FUNCTION_BLOCK FB_LightOffCommand IMPLEMENTS I_Command
VAR_INPUT
END_VAR
VAR_OUTPUT
END_VAR
VAR
	// Reference to the Light that should be switched on.
	iLight: I_Switchable;
END_VAR

METHOD Execute
IF (iLight <> 0) THEN
	THIS^.iLight.Off();
END_IF
END_METHOD

METHOD FB_init : BOOL
VAR_INPUT
	bInitRetains : BOOL; // if TRUE, the retain variables are initialized (warm start / cold start)
	bInCopyCode : BOOL;  // if TRUE, the instance afterwards gets moved into the copy code (online change)
	iSwitchable : I_Switchable;
END_VAR
IF (iSwitchable <> 0) THEN
	THIS^.iLight := iSwitchable;
END_IF
END_METHOD

END_FUNCTION_BLOCK

(* stored: Version 1.1.0.1, ProductVersion 3.1.4024.5
   POU FB_LightOffCommand: Id {fe928a09-9458-44e0-9164-25e795f97c63}, SpecialFunc None
   Method Execute: Id {e567bd74-9075-4f0a-81a2-b41c5c251ebd}
   Method FB_init: Id {a6205832-a0a7-4df8-92c1-8182aba049aa} *)
